{attribute 'qualified_only'}
VAR_GLOBAL
		Encoder_Counts AT %I* : UINT;
END_VAR

(* stored: Version 1.1.0.1, ProductVersion 3.1.4024.15
   GVL GVL_IO: Id {2134f0c0-7bc7-41e7-93e4-4b90a1ce6edf} *)
